Staubli VAL3: onInsert.pgx

public program onInsert(string& x_sItem[])
  local num l_nDelay
begin
  cls()
  l_nDelay=0
  call use:insertDialog("Distance [mm] ",l_nDelay,-0.01,2680.01)
  // give back
  if l_nDelay>=0
    l_nDelay=round(l_nDelay)
    x_sItem="AXISMOVEL "+toString("",l_nDelay)
  endIf
end
